// TIA Portal project "2022.09.06-步进电机往返运动仿真" (V17)

(* hardware
DEVICE "HMI_1"  KTP700 Basic PN
   slot 0: "HMI_1"  KTP700 Basic PN  6AV2 123-2GB03-0AX0  15.1.0.0
   slot 1: "HMI_RT_1"  KTP700 Basic PN  6AV2 123-2GB03-0AX0  15.1.0.0
   slot 5: "HMI_1.IE_CP_1"  PROFINET Interface  15.0.1.0
      slot 1: "PROFINET Interface_1"  PROFINET Interface
         slot 1: "Port_1"  Port
DEVICE "S7-1200 station_1"  S7-1200 Station
   slot 0: "Rack_0"  S7-1200 Rack  Rack  V1.0
   slot 1: "PLC_1"  CPU 1214C DC/DC/Rly  6ES7 214-1HG40-0XB0  V4.2
*)

// ===== PLC "PLC_1"  CPU 1214C DC/DC/Rly =====

VAR_GLOBAL   // PLC tag table "默认变量表"
   "轴1_脉冲" AT %Q0.3 : Bool;
   "轴1_方向" AT %Q0.4 : Bool;
   "轴1_归为开关" AT %Q0.2 : Bool;
   "轴复位" AT %M10.4 : Bool;
   "轴前进" AT %M10.5 : Bool;
   "轴后退" AT %M10.6 : Bool;
   "启动" AT %M0.0 : Bool;
   "停止" AT %M0.1 : Bool;
   "左限位" AT %I0.1 : Bool;
   "右限位" AT %I0.2 : Bool;
   "点动运行" AT %M11.3 : Bool;
   "相对位移启动" AT %M11.1 : Bool;
   "位移速度" AT %MD20 : Real;
   "相对位移速度" AT %MD24 : Real;
   "相对位移距离" AT %MD28 : Real;
   "轴_1_归位开关" AT %I0.3 : Bool;
   "Tag_1" AT %M11.0 : Bool;
   "Tag_2" AT %M10.7 : Bool;
   "Tag_3" AT %M110.0 : Bool;
   "Tag_4" AT %M10.0 : Bool;
   "Tag_5" AT %M10.1 : Bool;
   "Tag_6" AT %M10.2 : Bool;
   "Tag_7" AT %M0.2 : Bool;
   "轴_1_脉冲" AT %Q0.0 : Bool;
   "轴_1_方向" AT %Q0.1 : Bool;
END_VAR

DATA_BLOCK "轴1"   // DB1, Motion_DB
{ S7_Optimized_Access := 'TRUE' }
AUTHOR : SIMATIC
FAMILY : BasicMC
NAME : TO_PosAx
VERSION : 6.0
// stored: InstanceOfName TO_PositioningAxis
"TO_PositioningAxis"
BEGIN
   // Axis.DirectionOutputEnabledCU = TRUE
   // Axis.SelectedChannel2EnumCU = %Q0.1
   // Axis.SelectedChannel1EnumCU = %Q0.0
   // Axis.HomingReferencePointSwitch_AddressCU = %I0.3
   // Axis.OnlinePtoModeCU = 16#0000_0002
   // Pulse.MinDeltaDeltaFrequencyCU = 0.004
   // Pulse.MaxDeltaDeltaFrequencyCU = 1.0E+10
   // Pulse.MinDeltaFrequencyCU = 0.005
   // Pulse.MaxDeltaFrequencyCU = 9.5E+9
   // Pulse.MinFrequencyCU = 1.0
   // Pulse.MaxFrequencyCU = 100000.0
   // Pulse.OutputSourceCU = 16#0000_0000
   // Axis.SelectPTO = 0
END_DATA_BLOCK

DATA_BLOCK "轴_1"   // DB8, Motion_DB
{ S7_Optimized_Access := 'TRUE' }
AUTHOR : SIMATIC
FAMILY : BasicMC
NAME : TO_PosAx
VERSION : 6.0
// stored: InstanceOfName TO_PositioningAxis
"TO_PositioningAxis"
BEGIN
   // Axis.OnlinePtoModeCU = 16#0000_0002
   // Axis.DirectionOutputEnabledCU = TRUE
   // Axis.SelectedChannel2EnumCU = %Q0.1
   // Axis.SelectedChannel1EnumCU = %Q0.0
   // Pulse.MinDeltaDeltaFrequencyCU = 0.004
   // Pulse.MaxDeltaDeltaFrequencyCU = 1.0E+10
   // Pulse.MinDeltaFrequencyCU = 0.005
   // Pulse.MaxDeltaFrequencyCU = 9.5E+9
   // Pulse.MinFrequencyCU = 1.0
   // Pulse.MaxFrequencyCU = 100000.0
   // Pulse.OutputSourceCU = 16#0000_0000
   // Axis.SelectPTO = 0
END_DATA_BLOCK

ORGANIZATION_BLOCK "Main"   // OB1, LAD, ProgramCycle
TITLE = "Main Program Sweep (Cycle)"
{ S7_Optimized_Access := 'TRUE' }
VERSION : 0.1
   VAR_INPUT
      Initial_Call : Bool;   // Initial call of this OB
      Remanence : Bool;   // =True, if remanent data are available
   END_VAR
BEGIN

REGION Network 1: 启动
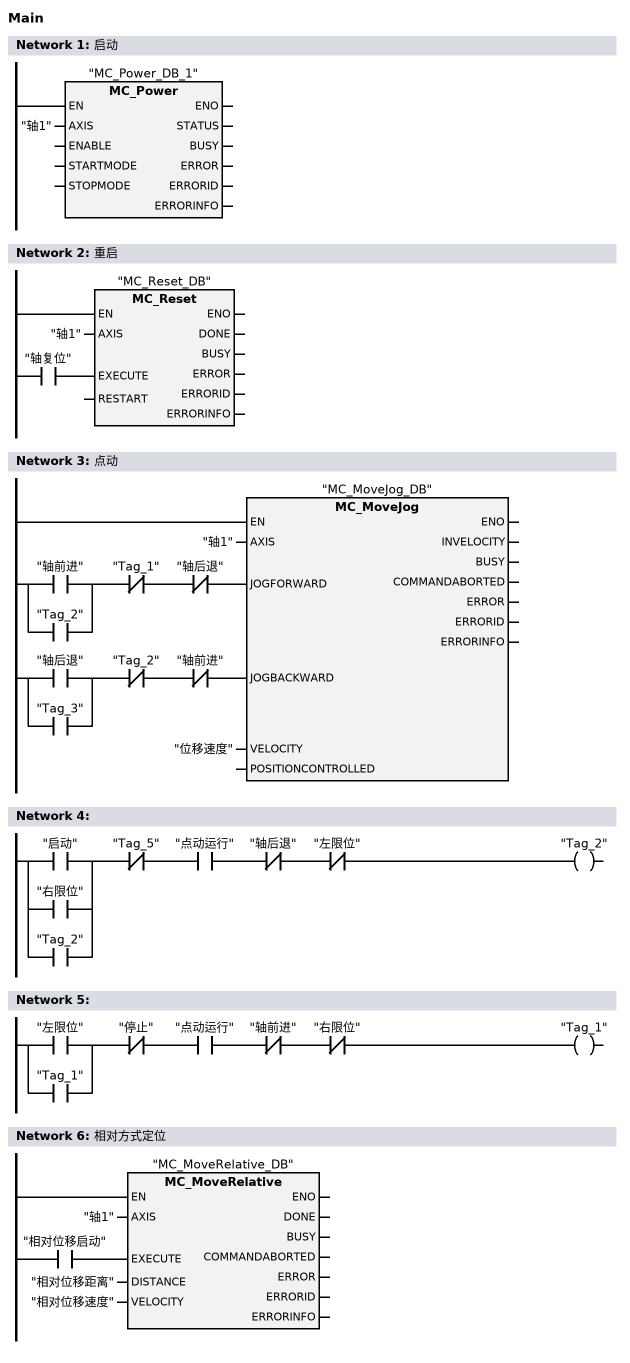
   "MC_Power_DB_1"(Axis := "轴1");   // MC_Power
END_REGION

REGION Network 2: 重启
   "MC_Reset_DB"(Axis := "轴1", Execute := "轴复位");   // MC_Reset
END_REGION

REGION Network 3: 点动
   "MC_MoveJog_DB"(Axis := "轴1",   // MC_MoveJog
                   JogForward := ("轴前进" OR "Tag_2") AND NOT "Tag_1" AND NOT "轴后退",
                   JogBackward := ("轴后退" OR "Tag_3") AND NOT "Tag_2" AND NOT "轴前进",
                   Velocity := "位移速度");
END_REGION

REGION Network 4
   RUNG wire#powerrail
      Contact( "启动" )
      wire#w1
      I_Contact( "Tag_5" )
      Contact( "点动运行" )
      I_Contact( "轴后退" )
      I_Contact( "左限位" )
      Coil( "Tag_2" )
   END_RUNG
   RUNG wire#powerrail
      Contact( "右限位" )
   END_RUNG wire#w1
   RUNG wire#powerrail
      Contact( "Tag_2" )
   END_RUNG wire#w1
   // the same network as SCL:
   "Tag_2" := ("启动" OR "右限位" OR "Tag_2") AND NOT "Tag_5" AND "点动运行" AND NOT "轴后退" AND NOT "左限位";
END_REGION

REGION Network 5
   RUNG wire#powerrail
      Contact( "左限位" )
      wire#w1
      I_Contact( "停止" )
      Contact( "点动运行" )
      I_Contact( "轴前进" )
      I_Contact( "右限位" )
      Coil( "Tag_1" )
   END_RUNG
   RUNG wire#powerrail
      Contact( "Tag_1" )
   END_RUNG wire#w1
   // the same network as SCL:
   "Tag_1" := ("左限位" OR "Tag_1") AND NOT "停止" AND "点动运行" AND NOT "轴前进" AND NOT "右限位";
END_REGION

REGION Network 6: 相对方式定位
   "MC_MoveRelative_DB"(Axis := "轴1", Execute := "相对位移启动", Distance := "相对位移距离", Velocity := "相对位移速度");   // MC_MoveRelative
END_REGION
END_ORGANIZATION_BLOCK

(* ===== HMI "HMI_RT_1" =====
system functions are stored by id; their names below are inferred from use
connection "HMI_连接_1": ETHERNET, SMART_S7_1200_OMS

HMI tags "默认变量表"
   "启动" : Bool = PLC 启动 AT %M0.0, 1 s
   "停止" : Bool = PLC 停止 AT %M0.1, 1 s
   "轴前进" : Bool = PLC 轴前进 AT %M10.5, 1 s
   "轴后退" : Bool = PLC 轴后退 AT %M10.6, 1 s
   "相对位移启动" : Bool = PLC 相对位移启动 AT %M11.1, 1 s
   "点动运行" : Bool = PLC 点动运行 AT %M11.3, 1 s
   "相对位移速度" : Real = PLC 相对位移速度 AT %MD24, 1 s
   "相对位移距离" : Real = PLC 相对位移距离 AT %MD28, 1 s
   "位移速度" : Real = PLC 位移速度 AT %MD20, 1 s

screen "画面_1" 800x480
   TextField "文本域_1" at 81,93 size 101x27; Text '循环位移'
   TextField "文本域_2" at 82,158 size 101x27; Text '点动位移'
   TextField "文本域_3" at 82,237 size 101x27; Text '相对位移'
   TextField "文本域_4" at 331,239 size 149x27; Text '相对位移距离'
   TextField "文本域_5" at 511,130 size 101x27; Text '点动速度'
   TextField "文本域_6" at 493,237 size 149x27; Text '相对位移速度'
   Button "按钮_1" at 201,85 size 96x32; TextOff '启动'
      on Press: SetBit("启动")
      on Release: ResetBit("启动")
   Button "按钮_2" at 200,153 size 96x32; TextOff '点动前进'
      on Release: ResetBit("轴前进")
      on Press: SetBit("轴前进")
   Button "按钮_3" at 201,234 size 107x32; TextOff '相对位移启动'
      on Release: ResetBit("相对位移启动")
      on Press: SetBit("相对位移启动")
   Button "按钮_4" at 351,85 size 96x32; TextOff '停止'
      on Press: SetBit("停止")
      on Release: ResetBit("停止")
   Button "按钮_5" at 351,153 size 96x32; TextOff '点动后退'
      on Press: SetBit("轴后退")
      on Release: ResetBit("轴后退")
   Button "按钮_6" at 500,86 size 130x32; TextOff '点动/循环往返'
      on Click: InvertBit("点动运行")
   TextField "文本域_7" at 179,14 size 269x37; Text '步进电机往返运动'
   IOField "I/O 域_1" at 341,275 size 131x56; FormatPattern s9999
      ProcessValue <- "相对位移距离"
   IOField "I/O 域_2" at 504,275 size 131x56; FormatPattern 99.9
      ProcessValue <- "相对位移速度"
   IOField "I/O 域_3" at 501,168 size 131x56; FormatPattern 99.9
      ProcessValue <- "位移速度"
   TextField "文本域_8" at 436,290 size 27x23; Text 'mm'
   TextField "文本域_9" at 578,183 size 49x23; Text 'mm/s'
   TextField "文本域_10" at 579,290 size 49x23; Text 'mm/s'
*)